PROGRAM Slit_3
VAR
    NorthSouthPowerOutput AT %Q* : BOOL:= TRUE;
    EastWestPowerOutput AT %Q* : BOOL:= TRUE;
END_VAR

END_PROGRAM

(* stored: Version 1.1.0.1, ProductVersion 3.1.4024.11
   POU Slit_3: Id {2442a95e-730f-4c91-8d13-516744e93144}, SpecialFunc None *)
